INTERFACE ITF_Component_HMI_Init EXTENDS ITF_BaseComponent, ITF_Component_HMI_Connector

END_INTERFACE

(* stored: Version 1.1.0.1, ProductVersion 3.1.4024.15
   Itf ITF_Component_HMI_Init: Id {87151dac-0541-41bf-9aff-bf7a6d50f3b8} *)
